# EPICS autosave request: support/ebrick/2-2-3/iocBoot/iocebrick/autosave/ebrickBRDADC.req
$(P)$(H)$(F)gain.VAL
$(P)$(H)$(F)gain.DESC
